{attribute 'GeneratedUsingTerminal: EL3318-0000-0016'}
{attribute addProperty BoxType "EL3318-0000-0016"}
{attribute addProperty Description "EL3318 8Ch. Ana Input Thermocouple (TC)"}
{attribute addProperty Physics "KK"}
{attribute addProperty Id "TC_Channel_1AT %I*TC_Channel_9575FEA17TC_Channel_2AT %I*TC_Channel_9575FEA17TC_Channel_3AT %I*TC_Channel_9575FEA17TC_Channel_4AT %I*TC_Channel_9575FEA17TC_Channel_5AT %I*TC_Channel_9575FEA17TC_Channel_6AT %I*TC_Channel_9575FEA17TC_Channel_7AT %I*TC_Channel_9575FEA17TC_Channel_8AT %I*TC_Channel_9575FEA17WcStateAT %I*WcState_9091E0EB2InfoDataAT %I*InfoData_32EB74EA10"}
{attribute addProperty CRC "1153518076"}
{attribute addProperty Size "68"}
TYPE EL3318_44C149FC EXTENDS EtcSlaveTerminalBase_947E5A46 :
STRUCT
	{attribute addProperty Name "TC_Channel_1"}
	TC_Channel_1 : TC_Channel_9575FEA1;
	{attribute addProperty Name "TC_Channel_2"}
	TC_Channel_2 : TC_Channel_9575FEA1;
	{attribute addProperty Name "TC_Channel_3"}
	TC_Channel_3 : TC_Channel_9575FEA1;
	{attribute addProperty Name "TC_Channel_4"}
	TC_Channel_4 : TC_Channel_9575FEA1;
	{attribute addProperty Name "TC_Channel_5"}
	TC_Channel_5 : TC_Channel_9575FEA1;
	{attribute addProperty Name "TC_Channel_6"}
	TC_Channel_6 : TC_Channel_9575FEA1;
	{attribute addProperty Name "TC_Channel_7"}
	TC_Channel_7 : TC_Channel_9575FEA1;
	{attribute addProperty Name "TC_Channel_8"}
	TC_Channel_8 : TC_Channel_9575FEA1;
	{attribute addProperty Name "WcState"}
	WcState : WcState_9091E0EB;
	{attribute addProperty Name "InfoData"}
	InfoData : InfoData_32EB74EA;
END_STRUCT
END_TYPE

(* stored: Version 1.2.0.0, ProductVersion 3.1.4024.9
   DUT EL3318_44C149FC: Id {78a5d8b0-fd3e-49ab-bb0b-75d06cd23e85} *)
